Fanuc KAREL source: kb00009.KL

PROGRAM KB00009
%STACKSIZE=65535
%PRIORITY=65535
%NOLOCKGROUP
VAR
P1 : REAL
P2 : REAL
RESULT : REAL
BEGIN
P1=1.0
P2=1.0
-- UNRESOLVED_PC line 10 opcodes [27 22 22 76 23] marker_code=32
END KB00009
